Universal Robots PolyScope program: LE03 RunTest 01.urp

Program LE03 RunTest 01 (installation=BK1 directory=/programs/LE createdIn=5.9.1.1031110 lastSavedIn=5.9.1.1031110 robotSerialNumber=20195501059)
Calibrated DH parameters: a=[0.000146, -0.418764, -0.053981, 0.000058, -0.000023, 0]; d=[0.162545, 37.319448, -206.067439, 168.881546, 0.09955, 0.099464]; alpha=[1.57004, -0.001979, 0.002304, 1.570607, -1.57066, 0]; deltaTheta=[0, -0.174616, -1.258233, 1.432844, -0.000001, 0]
BeforeStart
  URCap Gripper Activate (Robotiq_Grippers, Robotiq Inc.) dataModel(ResetAndActivateKey=false)
  URCap Gripper (Robotiq_Grippers, Robotiq Inc.) dataModel(position=100.0, force=100.0, speed=100.0, positionInDouble=100.0, forceInDouble=100.0, speedInDouble=100.0, slaveIds=[9], blocking=true)
  start_pose := get_actual_tcp_pose()
  MoveJ speed 60 deg/s, acceleration 80 deg/s^2 (useActiveTCP=true) feature=Base
    Waypoint Waypoint (Variable): variable=start_pose
Robot Program (runOnlyOnce=true)
  '2F85 Tool vertical above box'
  MoveJ speed 60 deg/s, acceleration 80 deg/s^2 (useActiveTCP=false) tcp=TCP_2F85; feature=Base
    Waypoint image_pose: TCP in base x=299.992 y=-399.925 z=99.974 mm, rx=0.0001 ry=0.0001 rz=0 rad; joints [111.361, -83.139, 115.497, -122.341, 270.047, 201.382] deg; TCP offset x=0 y=0 z=175 mm, rx=3.1416 ry=0 rz=0 rad
  MoveL speed 250 mm/s, acceleration 1200 mm/s^2 (useActiveTCP=false) tcp=TCP_2F85; feature=Base
    Waypoint on_target: TCP in base x=299.979 y=-399.967 z=4.98 mm, rx=0.0001 ry=0.0001 rz=0.0001 rad; joints [111.351, -73.735, 121.602, -137.854, 270.051, 201.396] deg
    Call move_on_axis
    Waypoint image_pose: TCP in base x=299.992 y=-399.925 z=99.974 mm, rx=0.0001 ry=0.0001 rz=0 rad; joints [111.361, -83.139, 115.497, -122.341, 270.047, 201.382] deg
  MoveL speed 250 mm/s, acceleration 1200 mm/s^2 (useActiveTCP=false) tcp=TCP_Basler; feature=Base
    Waypoint on_target: TCP in base x=299.979 y=-399.967 z=4.98 mm, rx=0.0001 ry=0.0001 rz=0.0001 rad; joints [111.351, -73.735, 121.602, -137.854, 270.051, 201.396] deg
    Call move_on_axis
    Waypoint image_pose: TCP in base x=299.992 y=-399.925 z=99.974 mm, rx=0.0001 ry=0.0001 rz=0 rad; joints [111.361, -83.139, 115.497, -122.341, 270.047, 201.382] deg
  MoveL speed 250 mm/s, acceleration 1200 mm/s^2 (useActiveTCP=false) tcp=TCP_Keyence; feature=Base
    Waypoint on_target: TCP in base x=299.979 y=-399.967 z=4.98 mm, rx=0.0001 ry=0.0001 rz=0.0001 rad; joints [111.351, -73.735, 121.602, -137.854, 270.051, 201.396] deg
    Call move_on_axis
    Waypoint image_pose: TCP in base x=299.992 y=-399.925 z=99.974 mm, rx=0.0001 ry=0.0001 rz=0 rad; joints [111.361, -83.139, 115.497, -122.341, 270.047, 201.382] deg
  MoveL speed 250 mm/s, acceleration 1200 mm/s^2 (useActiveTCP=false) tcp=TCP_2F85; feature=Base
    Waypoint image_pose: TCP in base x=299.992 y=-399.925 z=99.974 mm, rx=0.0001 ry=0.0001 rz=0 rad; joints [111.361, -83.139, 115.497, -122.341, 270.047, 201.382] deg
SubProgram -> move_on_axis
SubProgram move_on_axis (keepSynchronizedWithDisk=false)
  MoveL speed 250 mm/s, acceleration 1200 mm/s^2 (useActiveTCP=true) feature=Base
    MoveDirectionNode (selectedDirection=ZPlus) feature=Joint_6_name
      Until DISTANCE (allowActions=false deceleration=3 distanceNodeType=STOP) Distance=0.05; motionParameters(blendRadius=0)
    MoveDirectionNode (selectedDirection=ZMinus) feature=Joint_6_name
      Until DISTANCE (allowActions=false deceleration=3 distanceNodeType=STOP) Distance=0.05; motionParameters(blendRadius=0)
    MoveDirectionNode (selectedDirection=ZPlus) feature=Joint_6_name
      Until DISTANCE (allowActions=false deceleration=3 distanceNodeType=STOP) Distance=0.025; motionParameters(blendRadius=0)
